Staubli VAL3: writeSingle.pgx

public program writeSingle(num x_nModuleId, num x_nPin, bool x_bState, bool& x_bSuccess)
  local dio l_diSignal
  local num l_nPins
begin
  // Copyright (c) 2021, Institute for Factory Automation and Production Systems (FAPS)
  //
  // Licensed under the Apache License, Version 2.0 (the "License");
  // you may not use this file except in compliance with the License.
  // You may obtain a copy of the License at
  //
  //     http://www.apache.org/licenses/LICENSE-2.0
  //
  // Unless required by applicable law or agreed to in writing, software
  // distributed under the License is distributed on an "AS IS" BASIS,
  // WITHOUT WARRANTIES OR CONDITIONS OF ANY KIND, either express or implied.
  // See the License for the specific language governing permissions and
  // limitations under the License.


  x_bSuccess=true

  // get max pin count for given module
  switch x_nModuleId
    case IOModule:USER_IN,IOModule:VALVE_OUT
      l_nPins=2
    break
    default
      x_bSuccess=false
    break
  endSwitch

  // return if unknown module id was given
  if (x_bSuccess==false)
    popUpMsg("Error! Unknown module id: "+toString("",x_nModuleId))
    return
  endIf

  // check if pin index is out of range
  if (x_nPin>=l_nPins)
    popUpMsg("Error! Trying to set pin "+toString("",x_nPin)+" of module "+toString("",x_nModuleId))
    x_bSuccess=false
    return
  endIf

  // link signal source to local variable if possible
  switch x_nModuleId
    case IOModule:VALVE_OUT
      dioLink(l_diSignal,diValveOut[x_nPin])
    break
  endSwitch

  // set dio if linked successfully
  if (x_bSuccess)
    l_diSignal=x_bState
  endIf

end
